    boolExpected : BOOL;
    boolActual : BOOL;
    byteExpected : BYTE;
    byteActual : BYTE;
    dateExpected : DATE;
    dateActual : DATE;
    dateAndTimeExpected : DATE_AND_TIME;
    dateAndTimeActual : DATE_AND_TIME;
    dintExpected : DINT;
    dintActual : DINT;
    dwordExpected : DWORD;
    dwordActual : DWORD;
    intExpected : INT;
    intActual : INT;
    lintExpected : LINT;
    lintActual : LINT;
    lrealExpected : LREAL;
    lrealActual : LREAL;
    ltimeExpected : LTIME;
    ltimeActual : LTIME;
    lwordExpected : LWORD;
    lwordActual : LWORD;
    realExpected : REAL;
    realActual : REAL;
    sintExpected : SINT;
    sintActual : SINT;
    stringExpected : Tc2_System.T_MaxString;
    stringActual : Tc2_System.T_MaxString;
    timeExpected : TIME;
    timeActual : TIME;
    timeOfDayExpected : TIME_OF_DAY;
    timeOfDayActual : TIME_OF_DAY;
    udintExpected : UDINT;
    udintActual : UDINT;
    uintExpected : UINT;
    uintActual : UINT;
    ulintExpected : ULINT;
    ulintActual : ULINT;
    usintExpected : USINT;
    usintActual : USINT;
    wordExpected : WORD;
    wordActual : WORD;
END_VAR
IF GVL_TcUnit.IgnoreCurrentTest OR GVL_TcUnit.CurrentTestIsFinished THEN
    RETURN;
END_IF

AnyComparator(AnyValueOne := Expected,
              AnyValueTwo := Actual);

(* First check whether the input data are any of the standard data types that are supported by TcUnit.
   In this case call the standard Assert-methods for that data. But before doing that we need to make sure
   that both the expected and actual:
   - Have both the same data type
   - Both have the same data size
*)
IF NOT AnyComparator.DataTypesNotEquals AND NOT AnyComparator.DataSizeNotEquals THEN

    (* BOOL *)
    IF UDINT_TO_INT(Expected.TypeClass) = IBaseLibrary.TypeClass.TYPE_BOOL THEN
        Tc2_System.MEMCPY(destAddr := ADR(boolExpected), srcAddr := Expected.pValue, n := SIZEOF(BOOL));
        Tc2_System.MEMCPY(destAddr := ADR(boolActual), srcAddr := Actual.pValue, n := SIZEOF(BOOL));
        AssertEquals_BOOL(Expected := boolExpected, Actual := boolActual, Message := Message);
        RETURN;
    END_IF

    (* BYTE *)
    IF UDINT_TO_INT(Expected.TypeClass) = IBaseLibrary.TypeClass.TYPE_BYTE THEN
        Tc2_System.MEMCPY(destAddr := ADR(byteExpected), srcAddr := Expected.pValue, n := SIZEOF(BYTE));
        Tc2_System.MEMCPY(destAddr := ADR(byteActual), srcAddr := Actual.pValue, n := SIZEOF(BYTE));
        AssertEquals_BYTE(Expected := byteExpected, Actual := byteActual, Message := Message);
        RETURN;
    END_IF

    (* DATE *)
    IF UDINT_TO_INT(Expected.TypeClass) = IBaseLibrary.TypeClass.TYPE_DATE THEN
        Tc2_System.MEMCPY(destAddr := ADR(dateExpected), srcAddr := Expected.pValue, n := SIZEOF(DATE));
        Tc2_System.MEMCPY(destAddr := ADR(dateActual), srcAddr := Actual.pValue, n := SIZEOF(DATE));
        AssertEquals_DATE(Expected := dateExpected, Actual := dateActual, Message := Message);
        RETURN;
    END_IF

    (* DATE_AND_TIME *)
    IF UDINT_TO_INT(Expected.TypeClass) = IBaseLibrary.TypeClass.TYPE_DATEANDTIME THEN
        Tc2_System.MEMCPY(destAddr := ADR(dateAndTimeExpected), srcAddr := Expected.pValue, n := SIZEOF(DATE_AND_TIME));
        Tc2_System.MEMCPY(destAddr := ADR(dateAndTimeActual), srcAddr := Actual.pValue, n := SIZEOF(DATE_AND_TIME));
        AssertEquals_DATE_AND_TIME(Expected := dateAndTimeExpected, Actual := dateAndTimeActual, Message := Message);
        RETURN;
    END_IF

    (* DINT *)
    IF UDINT_TO_INT(Expected.TypeClass) = IBaseLibrary.TypeClass.TYPE_DINT THEN
        Tc2_System.MEMCPY(destAddr := ADR(dintExpected), srcAddr := Expected.pValue, n := SIZEOF(DINT));
        Tc2_System.MEMCPY(destAddr := ADR(dintActual), srcAddr := Actual.pValue, n := SIZEOF(DINT));
        AssertEquals_DINT(Expected := dintExpected, Actual := dintActual, Message := Message);
        RETURN;
    END_IF

    (* DWORD *)
    IF UDINT_TO_INT(Expected.TypeClass) = IBaseLibrary.TypeClass.TYPE_DWORD THEN
        Tc2_System.MEMCPY(destAddr := ADR(dwordExpected), srcAddr := Expected.pValue, n := SIZEOF(DWORD));
        Tc2_System.MEMCPY(destAddr := ADR(dwordActual), srcAddr := Actual.pValue, n := SIZEOF(DWORD));
        AssertEquals_DWORD(Expected := dwordExpected, Actual := dwordActual, Message := Message);
        RETURN;
    END_IF

    (* INT *)
    IF UDINT_TO_INT(Expected.TypeClass) = IBaseLibrary.TypeClass.TYPE_INT THEN
        Tc2_System.MEMCPY(destAddr := ADR(intExpected), srcAddr := Expected.pValue, n := SIZEOF(INT));
        Tc2_System.MEMCPY(destAddr := ADR(intActual), srcAddr := Actual.pValue, n := SIZEOF(INT));
        AssertEquals_INT(Expected := intExpected, Actual := intActual, Message := Message);
        RETURN;
    END_IF

    (* LINT *)
    IF UDINT_TO_INT(Expected.TypeClass) = IBaseLibrary.TypeClass.TYPE_LINT THEN
        Tc2_System.MEMCPY(destAddr := ADR(lintExpected), srcAddr := Expected.pValue, n := SIZEOF(LINT));
        Tc2_System.MEMCPY(destAddr := ADR(lintActual), srcAddr := Actual.pValue, n := SIZEOF(LINT));
        AssertEquals_LINT(Expected := lintExpected, Actual := lintActual, Message := Message);
        RETURN;
    END_IF

    (* LREAL *)
    IF UDINT_TO_INT(Expected.TypeClass) = IBaseLibrary.TypeClass.TYPE_LREAL THEN
        Tc2_System.MEMCPY(destAddr := ADR(lrealExpected), srcAddr := Expected.pValue, n := SIZEOF(LREAL));
        Tc2_System.MEMCPY(destAddr := ADR(lrealActual), srcAddr := Actual.pValue, n := SIZEOF(LREAL));
        AssertEquals_LREAL(Expected := lrealExpected, Actual := lrealActual, Delta := 0.0, Message := Message);
        RETURN;
    END_IF

    (* LTIME *)
    IF UDINT_TO_INT(Expected.TypeClass) = IBaseLibrary.TypeClass.TYPE_LTIME THEN
        Tc2_System.MEMCPY(destAddr := ADR(ltimeExpected), srcAddr := Expected.pValue, n := SIZEOF(LTIME));
        Tc2_System.MEMCPY(destAddr := ADR(ltimeActual), srcAddr := Actual.pValue, n := SIZEOF(LTIME));
        AssertEquals_LTIME(Expected := ltimeExpected, Actual := ltimeActual, Message := Message);
        RETURN;
    END_IF

    (* LWORD *)
    IF UDINT_TO_INT(Expected.TypeClass) = IBaseLibrary.TypeClass.TYPE_LWORD THEN
        Tc2_System.MEMCPY(destAddr := ADR(lwordExpected), srcAddr := Expected.pValue, n := SIZEOF(LWORD));
        Tc2_System.MEMCPY(destAddr := ADR(lwordActual), srcAddr := Actual.pValue, n := SIZEOF(LWORD));
        AssertEquals_LWORD(Expected := lwordExpected, Actual := lwordActual, Message := Message);
        RETURN;
    END_IF

    (* REAL *)
    IF UDINT_TO_INT(Expected.TypeClass) = IBaseLibrary.TypeClass.TYPE_REAL THEN
        Tc2_System.MEMCPY(destAddr := ADR(realExpected), srcAddr := Expected.pValue, n := SIZEOF(REAL));
        Tc2_System.MEMCPY(destAddr := ADR(realActual), srcAddr := Actual.pValue, n := SIZEOF(REAL));
        AssertEquals_REAL(Expected := realExpected, Actual := realActual, Delta := 0.0, Message := Message);
        RETURN;
    END_IF

    (* SINT *)
    IF UDINT_TO_INT(Expected.TypeClass) = IBaseLibrary.TypeClass.TYPE_SINT THEN
        Tc2_System.MEMCPY(destAddr := ADR(sintExpected), srcAddr := Expected.pValue, n := SIZEOF(SINT));
        Tc2_System.MEMCPY(destAddr := ADR(sintActual), srcAddr := Actual.pValue, n := SIZEOF(SINT));
        AssertEquals_SINT(Expected := sintExpected, Actual := sintActual, Message := Message);
        RETURN;
    END_IF

    (* STRING *)
    IF UDINT_TO_INT(Expected.TypeClass) = IBaseLibrary.TypeClass.TYPE_STRING THEN
        Tc2_System.MEMCPY(destAddr := ADR(stringExpected), srcAddr := Expected.pValue, n := DINT_TO_UDINT(Expected.diSize));
        Tc2_System.MEMCPY(destAddr := ADR(stringActual), srcAddr := Actual.pValue, n := DINT_TO_UDINT(Actual.diSize));
        AssertEquals_STRING(Expected := stringExpected, Actual := stringActual, Message := Message);
        RETURN;
    END_IF

    (* TIME *)
    IF UDINT_TO_INT(Expected.TypeClass) = IBaseLibrary.TypeClass.TYPE_TIME THEN
        Tc2_System.MEMCPY(destAddr := ADR(timeExpected), srcAddr := Expected.pValue, n := SIZEOF(TIME));
        Tc2_System.MEMCPY(destAddr := ADR(timeActual), srcAddr := Actual.pValue, n := SIZEOF(TIME));
        AssertEquals_TIME(Expected := timeExpected, Actual := timeActual, Message := Message);
        RETURN;
    END_IF

    (* TIME_OF_DAY *)
    IF UDINT_TO_INT(Expected.TypeClass) = IBaseLibrary.TypeClass.TYPE_TIMEOFDAY THEN
        Tc2_System.MEMCPY(destAddr := ADR(timeOfDayExpected), srcAddr := Expected.pValue, n := SIZEOF(TIME_OF_DAY));
        Tc2_System.MEMCPY(destAddr := ADR(timeOfDayActual), srcAddr := Actual.pValue, n := SIZEOF(TIME_OF_DAY));
        AssertEquals_TIME_OF_DAY(Expected := timeOfDayExpected, Actual := timeOfDayActual, Message := Message);
        RETURN;
    END_IF

    (* UDINT *)
    IF UDINT_TO_INT(Expected.TypeClass) = IBaseLibrary.TypeClass.TYPE_UDINT THEN
        Tc2_System.MEMCPY(destAddr := ADR(udintExpected), srcAddr := Expected.pValue, n := SIZEOF(UDINT));
        Tc2_System.MEMCPY(destAddr := ADR(udintActual), srcAddr := Actual.pValue, n := SIZEOF(UDINT));
        AssertEquals_UDINT(Expected := udintExpected, Actual := udintActual, Message := Message);
        RETURN;
    END_IF

    (* UINT *)
    IF UDINT_TO_INT(Expected.TypeClass) = IBaseLibrary.TypeClass.TYPE_UINT THEN
        Tc2_System.MEMCPY(destAddr := ADR(uintExpected), srcAddr := Expected.pValue, n := SIZEOF(UINT));
        Tc2_System.MEMCPY(destAddr := ADR(uintActual), srcAddr := Actual.pValue, n := SIZEOF(UINT));
        AssertEquals_UINT(Expected := uintExpected, Actual := uintActual, Message := Message);
        RETURN;
    END_IF

    (* ULINT *)
    IF UDINT_TO_INT(Expected.TypeClass) = IBaseLibrary.TypeClass.TYPE_ULINT THEN
        Tc2_System.MEMCPY(destAddr := ADR(ulintExpected), srcAddr := Expected.pValue, n := SIZEOF(ULINT));
        Tc2_System.MEMCPY(destAddr := ADR(ulintActual), srcAddr := Actual.pValue, n := SIZEOF(ULINT));
        AssertEquals_ULINT(Expected := ulintExpected, Actual := ulintActual, Message := Message);
        RETURN;
    END_IF

    (* USINT *)
    IF UDINT_TO_INT(Expected.TypeClass) = IBaseLibrary.TypeClass.TYPE_USINT THEN
        Tc2_System.MEMCPY(destAddr := ADR(usintExpected), srcAddr := Expected.pValue, n := SIZEOF(USINT));
        Tc2_System.MEMCPY(destAddr := ADR(usintActual), srcAddr := Actual.pValue, n := SIZEOF(USINT));
        AssertEquals_USINT(Expected := usintExpected, Actual := usintActual, Message := Message);
        RETURN;
    END_IF

    (* WORD *)
    IF UDINT_TO_INT(Expected.TypeClass) = IBaseLibrary.TypeClass.TYPE_WORD THEN
        Tc2_System.MEMCPY(destAddr := ADR(wordExpected), srcAddr := Expected.pValue, n := SIZEOF(WORD));
        Tc2_System.MEMCPY(destAddr := ADR(wordActual), srcAddr := Actual.pValue, n := SIZEOF(WORD));
        AssertEquals_WORD(Expected := wordExpected, Actual := wordActual, Message := Message);
        RETURN;
    END_IF

END_IF

(* If we've come to this row, it means that the data input is not any of the standard primitive data types, and thus
   we need to do special handling *)
TestInstancePath := AddTestNameToInstancePath(TestInstancePath := FindTestSuiteInstancePath());

IF AnyComparator.DataTypesNotEquals THEN
    ExpectedDataString := Tc2_Standard.CONCAT(STR1 := '(Type class = ', STR2 := F_AnyTypeClassToString((Expected.TypeClass)));
    ExpectedDataString := Tc2_Standard.CONCAT(STR1 := ExpectedDataString, STR2 := ')');
    ActualDataString := Tc2_Standard.CONCAT(STR1 := '(Type class = ', STR2 := F_AnyTypeClassToString(Actual.TypeClass));
    ActualDataString := Tc2_Standard.CONCAT(STR1 := ActualDataString, STR2 := ')');
ELSIF AnyComparator.DataSizeNotEquals THEN
    ExpectedDataString := Tc2_Standard.CONCAT(STR1 := '(Data size = ', STR2 := DINT_TO_STRING(Expected.diSize));
    ExpectedDataString := Tc2_Standard.CONCAT(STR1 := ExpectedDataString, STR2 := ')');
    ActualDataString := Tc2_Standard.CONCAT(STR1 := '(Data size = ', STR2 := DINT_TO_STRING(Actual.diSize));
    ActualDataString := Tc2_Standard.CONCAT(STR1 := ActualDataString, STR2 := ')');
ELSIF AnyComparator.DataContentNotEquals THEN
    FOR Count := 0 TO MIN(Expected.diSize-1, 38) BY 1 DO // One byte will equal two characters (example: 255 = 0xff, 1 = 0x01)
        ExpectedDataString := Tc2_Standard.CONCAT(STR1 := ExpectedDataString,
                                                  STR2 := Tc2_Utilities.BYTE_TO_HEXSTR(in := Expected.pValue[Count],
                                                                                       iPrecision := 2,
                                                                                       bLoCase := FALSE));
    END_FOR
    ExpectedDataString := Tc2_Standard.CONCAT(STR1 := '0x', STR2 := ExpectedDataString);

    FOR Count := 0 TO MIN(Actual.diSize-1, 38) BY 1 DO // One byte will equal two characters (example: 255 = 0xff, 1 = 0x01)
        ActualDataString := Tc2_Standard.CONCAT(STR1 := ActualDataString,
                                                STR2 := Tc2_Utilities.BYTE_TO_HEXSTR(in := Actual.pValue[Count],
                                                                                     iPrecision := 2,
                                                                                     bLoCase := FALSE));
    END_FOR
    ActualDataString := Tc2_Standard.CONCAT(STR1 := '0x', STR2 := ActualDataString);
END_IF

IF (AnyComparator.DataTypesNotEquals OR AnyComparator.DataSizeNotEquals OR AnyComparator.DataContentNotEquals) THEN
    AssertResults.ReportResult(Expected := Expected,
                               Actual := Actual,
                               Message := Message,
                               TestInstancePath := TestInstancePath,
                               AlreadyReported => AlreadyReported);
END_IF

IF NOT AlreadyReported AND (AnyComparator.DataTypesNotEquals OR AnyComparator.DataSizeNotEquals OR AnyComparator.DataContentNotEquals) THEN
    SetTestFailed();

    AssertMessageFormatter.LogAssertFailure(Expected := ExpectedDataString,
                                            Actual := ActualDataString,
                                            Message := Message,
                                            TestInstancePath := TestInstancePath);
END_IF
END_METHOD

(*
    Asserts that two BOOLs are equal. If they are not, an assertion error is created.
*)
METHOD PUBLIC AssertEquals_BOOL
VAR_INPUT
    Expected : BOOL; // BOOL expected value
    Actual : BOOL; // BOOL actual value
    Message : Tc2_System.T_MaxString; // The identifying message for the assertion error
END_VAR
VAR
    AlreadyReported : BOOL;
    TestInstancePath : Tc2_System.T_MaxString;
END_VAR
IF GVL_TcUnit.IgnoreCurrentTest OR GVL_TcUnit.CurrentTestIsFinished THEN
    RETURN;
END_IF

TestInstancePath := AddTestNameToInstancePath(TestInstancePath := FindTestSuiteInstancePath());

IF Expected <> Actual THEN
    AssertResults.ReportResult(Expected := Expected,
                               Actual := Actual,
                               Message := Message,
                               TestInstancePath := TestInstancePath,
                               AlreadyReported => AlreadyReported);
END_IF                               

IF NOT AlreadyReported AND Expected <> Actual THEN
    SetTestFailed();

    AssertMessageFormatter.LogAssertFailure(Expected := BOOL_TO_STRING(Expected),
                                            Actual := BOOL_TO_STRING(Actual),
                                            Message := Message,
                                            TestInstancePath := TestInstancePath);
END_IF
END_METHOD

(*
    Asserts that two BYTEs are equal. If they are not, an assertion error is created.
*)
METHOD PUBLIC AssertEquals_BYTE
VAR_INPUT
    Expected : BYTE; // BYTE expected value
    Actual : BYTE; // BYTE actual value
    Message : Tc2_System.T_MaxString; // The identifying message for the assertion error
END_VAR
VAR
    TestInstancePath : Tc2_System.T_MaxString;
    AlreadyReported : BOOL;
END_VAR
IF GVL_TcUnit.IgnoreCurrentTest OR GVL_TcUnit.CurrentTestIsFinished THEN
    RETURN;
END_IF

TestInstancePath := AddTestNameToInstancePath(TestInstancePath := FindTestSuiteInstancePath());

IF Expected <> Actual THEN
    AssertResults.ReportResult(Expected := Expected,
                               Actual := Actual,
                               Message := Message,
                               TestInstancePath := TestInstancePath,
                               AlreadyReported => AlreadyReported);
END_IF

IF NOT AlreadyReported AND Expected <> Actual THEN
    SetTestFailed();

    AssertMessageFormatter.LogAssertFailure(Expected := Tc2_Standard.CONCAT(
                                                       STR1 := '0x',
                                                       STR2 := Tc2_Utilities.BYTE_TO_HEXSTR(in := Expected,
                                                                                            iPrecision := 2,
                                                                                            bLoCase := FALSE)),
                                            Actual := Tc2_Standard.CONCAT(
                                                       STR1 := '0x',
                                                       STR2 := Tc2_Utilities.BYTE_TO_HEXSTR(in := Actual,
                                                                                            iPrecision := 2,
                                                                                            bLoCase := FALSE)),
                                            Message := Message,
                                            TestInstancePath := TestInstancePath);
END_IF
END_METHOD

(*
    Asserts that two DATEs are equal. If they are not, an assertion error is created.
*)
METHOD PUBLIC AssertEquals_DATE
VAR_INPUT
    Expected : DATE; // DATE expected value
    Actual : DATE; // DATE actual value
    Message : Tc2_System.T_MaxString; // The identifying message for the assertion error
END_VAR
VAR
    TestInstancePath : Tc2_System.T_MaxString;
    AlreadyReported : BOOL;
END_VAR
IF GVL_TcUnit.IgnoreCurrentTest OR GVL_TcUnit.CurrentTestIsFinished THEN
    RETURN;
END_IF

TestInstancePath := AddTestNameToInstancePath(TestInstancePath := FindTestSuiteInstancePath());

IF Expected <> Actual THEN
    AssertResults.ReportResult(Expected := Expected,
                               Actual := Actual,
                               Message := Message,
                               TestInstancePath := TestInstancePath,
                               AlreadyReported => AlreadyReported);
END_IF

IF NOT AlreadyReported AND Expected <> Actual THEN
    SetTestFailed();

    AssertMessageFormatter.LogAssertFailure(Expected := DATE_TO_STRING(Expected),
                                            Actual := DATE_TO_STRING(Actual),
                                            Message := Message,
                                            TestInstancePath := TestInstancePath);
END_IF
END_METHOD

(*
    Asserts that two DATE_AND_TIMEs are equal. If they are not, an assertion error is created.
*)
METHOD PUBLIC AssertEquals_DATE_AND_TIME
VAR_INPUT
    Expected : DATE_AND_TIME; // DATE_AND_TIME expected value
    Actual : DATE_AND_TIME; // DATE_AND_TIME actual value
    Message : Tc2_System.T_MaxString; // The identifying message for the assertion error
END_VAR
VAR
    TestInstancePath : Tc2_System.T_MaxString;
    AlreadyReported : BOOL;
END_VAR
IF GVL_TcUnit.IgnoreCurrentTest OR GVL_TcUnit.CurrentTestIsFinished THEN
    RETURN;
END_IF

TestInstancePath := AddTestNameToInstancePath(TestInstancePath := FindTestSuiteInstancePath());

IF Expected <> Actual THEN
    AssertResults.ReportResult(Expected := Expected,
                               Actual := Actual,
                               Message := Message,
                               TestInstancePath := TestInstancePath,
                               AlreadyReported => AlreadyReported);
END_IF

IF NOT AlreadyReported AND Expected <> Actual THEN
    SetTestFailed();

    AssertMessageFormatter.LogAssertFailure(Expected := DT_TO_STRING(Expected),
                                            Actual := DT_TO_STRING(Actual),
                                            Message := Message,
                                            TestInstancePath := TestInstancePath);
END_IF
END_METHOD

(*
    Asserts that two DINTs are equal. If they are not, an assertion error is created.
*)
METHOD PUBLIC AssertEquals_DINT
VAR_INPUT
    Expected : DINT; // DINT expected value
    Actual : DINT; // DINT actual value
    Message : Tc2_System.T_MaxString; // The identifying message for the assertion error
END_VAR
VAR
    TestInstancePath : Tc2_System.T_MaxString;
    AlreadyReported : BOOL;
END_VAR
IF GVL_TcUnit.IgnoreCurrentTest OR GVL_TcUnit.CurrentTestIsFinished THEN
    RETURN;
END_IF

TestInstancePath := AddTestNameToInstancePath(TestInstancePath := FindTestSuiteInstancePath());

IF Expected <> Actual THEN
    AssertResults.ReportResult(Expected := Expected,
                               Actual := Actual,
                               Message := Message,
                               TestInstancePath := TestInstancePath,
                               AlreadyReported => AlreadyReported);
END_IF

IF NOT AlreadyReported AND Expected <> Actual THEN
    SetTestFailed();

    AssertMessageFormatter.LogAssertFailure(Expected := DINT_TO_STRING(Expected),
                                            Actual := DINT_TO_STRING(Actual),
                                            Message := Message,
                                            TestInstancePath := TestInstancePath);
END_IF
END_METHOD

(*
    Asserts that two DWORDs are equal. If they are not, an assertion error is created.
*)
METHOD PUBLIC AssertEquals_DWORD
VAR_INPUT
    Expected : DWORD; // DWORD expected value
    Actual : DWORD; // DWORD actual value
    Message : Tc2_System.T_MaxString; // The identifying message for the assertion error
END_VAR
VAR
    TestInstancePath : Tc2_System.T_MaxString;
    AlreadyReported : BOOL;
END_VAR
IF GVL_TcUnit.IgnoreCurrentTest OR GVL_TcUnit.CurrentTestIsFinished THEN
    RETURN;
END_IF

TestInstancePath := AddTestNameToInstancePath(TestInstancePath := FindTestSuiteInstancePath());

IF Expected <> Actual THEN
    AssertResults.ReportResult(Expected := Expected,
                               Actual := Actual,
                               Message := Message,
                               TestInstancePath := TestInstancePath,
                               AlreadyReported => AlreadyReported);
END_IF

IF NOT AlreadyReported AND Expected <> Actual THEN
    SetTestFailed();

    AssertMessageFormatter.LogAssertFailure(Expected := Tc2_Standard.CONCAT(
                                                            STR1 := '0x',
                                                            STR2 := Tc2_Utilities.DWORD_TO_HEXSTR(in := Expected,
                                                                                                  iPrecision := 8,
                                                                                                  bLoCase := FALSE)),
                                            Actual := Tc2_Standard.CONCAT(
                                                           STR1 := '0x',
                                                           STR2 := Tc2_Utilities.DWORD_TO_HEXSTR(in := Actual,
                                                                                                 iPrecision := 8,
                                                                                                 bLoCase := FALSE)),
                                            Message := Message,
                                            TestInstancePath := TestInstancePath);
END_IF
END_METHOD

(*
    Asserts that two INTs are equal. If they are not, an assertion error is created.
*)
METHOD PUBLIC AssertEquals_INT
VAR_INPUT
    Expected : INT; // INT expected value
    Actual : INT; // INT actual value
    Message : Tc2_System.T_MaxString; // The identifying message for the assertion error
END_VAR
VAR
    TestInstancePath : Tc2_System.T_MaxString;
    AlreadyReported : BOOL;
END_VAR
IF GVL_TcUnit.IgnoreCurrentTest OR GVL_TcUnit.CurrentTestIsFinished THEN
    RETURN;
END_IF

TestInstancePath := AddTestNameToInstancePath(TestInstancePath := FindTestSuiteInstancePath());

IF Expected <> Actual THEN
    AssertResults.ReportResult(Expected := Expected,
                               Actual := Actual,
                               Message := Message,
                               TestInstancePath := TestInstancePath,
                               AlreadyReported => AlreadyReported);
END_IF

IF NOT AlreadyReported AND Expected <> Actual THEN
    SetTestFailed();

    AssertMessageFormatter.LogAssertFailure(Expected := INT_TO_STRING(Expected),
                                            Actual := INT_TO_STRING(Actual),
                                            Message := Message,
                                            TestInstancePath := TestInstancePath);
END_IF
END_METHOD

(*
    Asserts that two LINTs are equal. If they are not, an assertion error is created.
*)
METHOD PUBLIC AssertEquals_LINT
VAR_INPUT
    Expected : LINT; // LINT expected value
    Actual : LINT; // LINT actual value
    Message : Tc2_System.T_MaxString; // The identifying message for the assertion error
END_VAR
VAR
    TestInstancePath : Tc2_System.T_MaxString;
    AlreadyReported : BOOL;
END_VAR
IF GVL_TcUnit.IgnoreCurrentTest OR GVL_TcUnit.CurrentTestIsFinished THEN
    RETURN;
END_IF

TestInstancePath := AddTestNameToInstancePath(TestInstancePath := FindTestSuiteInstancePath());

IF Expected <> Actual THEN
    AssertResults.ReportResult(Expected := Expected,
                               Actual := Actual,
                               Message := Message,
                               TestInstancePath := TestInstancePath,
                               AlreadyReported => AlreadyReported);
END_IF

IF NOT AlreadyReported AND Expected <> Actual THEN
    SetTestFailed();

    AssertMessageFormatter.LogAssertFailure(Expected := LINT_TO_STRING(Expected),
                                            Actual := LINT_TO_STRING(Actual),
                                            Message := Message,
                                            TestInstancePath := TestInstancePath);
END_IF
END_METHOD

(*
    Asserts that two LREALs are equal to within a positive delta. If they are not, an assertion error is created.
*)
METHOD PUBLIC AssertEquals_LREAL
VAR_INPUT
    Expected : LREAL; // LREAL expected value
    Actual : LREAL; // LREAL actual value
    Delta : LREAL; // The maximum delta between the absolute value of expected and actual for which both numbers are still considered equal
    Message : Tc2_System.T_MaxString; // The identifying message for the assertion error
END_VAR
VAR
    TestInstancePath : Tc2_System.T_MaxString;
    AlreadyReported : BOOL;
END_VAR
IF GVL_TcUnit.IgnoreCurrentTest OR GVL_TcUnit.CurrentTestIsFinished THEN
    RETURN;
END_IF

TestInstancePath := AddTestNameToInstancePath(TestInstancePath := FindTestSuiteInstancePath());

IF ABS(Expected - Actual) > Delta THEN
    AssertResults.ReportResult(Expected := Expected,
                               Actual := Actual,
                               Message := Message,
                               TestInstancePath := TestInstancePath,
                               AlreadyReported => AlreadyReported);
END_IF

IF NOT AlreadyReported AND ABS(Expected - Actual) > Delta THEN
    SetTestFailed();

    AssertMessageFormatter.LogAssertFailure(Expected := LREAL_TO_STRING(Expected),
                                            Actual := LREAL_TO_STRING(Actual),
                                            Message := Message,
                                            TestInstancePath := TestInstancePath);
END_IF
END_METHOD

(*
    Asserts that two LTIMEs are equal. If they are not, an assertion error is created.
*)
METHOD PUBLIC AssertEquals_LTIME
VAR_INPUT
    Expected : LTIME; // LTIME expected value
    Actual : LTIME; // LTIME actual value
    Message : Tc2_System.T_MaxString; // The identifying message for the assertion error
END_VAR
VAR
    TestInstancePath : Tc2_System.T_MaxString;
    AlreadyReported : BOOL;
END_VAR
IF GVL_TcUnit.IgnoreCurrentTest OR GVL_TcUnit.CurrentTestIsFinished THEN
    RETURN;
END_IF

TestInstancePath := AddTestNameToInstancePath(TestInstancePath := FindTestSuiteInstancePath());

IF Expected <> Actual THEN
    AssertResults.ReportResult(Expected := Expected,
                               Actual := Actual,
                               Message := Message,
                               TestInstancePath := TestInstancePath,
                               AlreadyReported => AlreadyReported);
END_IF

IF NOT AlreadyReported AND Expected <> Actual THEN
    SetTestFailed();

    AssertMessageFormatter.LogAssertFailure(Expected := LTIME_TO_STRING(Expected),
                                            Actual := LTIME_TO_STRING(Actual),
                                            Message := Message,
                                            TestInstancePath := TestInstancePath);
END_IF
END_METHOD

(*
    Asserts that two LWORDs are equal. If they are not, an assertion error is created.
*)
METHOD PUBLIC AssertEquals_LWORD
VAR_INPUT
    Expected : LWORD; // LWORD expected value
    Actual : LWORD; // LWORD actual value
    Message : Tc2_System.T_MaxString; // The identifying message for the assertion error
END_VAR
VAR
    TestInstancePath : Tc2_System.T_MaxString;
    AlreadyReported : BOOL;
END_VAR
IF GVL_TcUnit.IgnoreCurrentTest OR GVL_TcUnit.CurrentTestIsFinished THEN
    RETURN;
END_IF

TestInstancePath := AddTestNameToInstancePath(TestInstancePath := FindTestSuiteInstancePath());

IF Expected <> Actual THEN
    AssertResults.ReportResult(Expected := Expected,
                               Actual := Actual,
                               Message := Message,
                               TestInstancePath := TestInstancePath,
                               AlreadyReported => AlreadyReported);
END_IF

IF NOT AlreadyReported AND Expected <> Actual THEN
    SetTestFailed();

    AssertMessageFormatter.LogAssertFailure(Expected := Tc2_Standard.CONCAT(
                                                            STR1 := '0x',
                                                            STR2 := Tc2_Utilities.LWORD_TO_HEXSTR(in := Expected,
                                                                                                  iPrecision := 16,
                                                                                                  bLoCase := FALSE)),
                                            Actual := Tc2_Standard.CONCAT(
                                                            STR1 := '0x',
                                                            STR2 := Tc2_Utilities.LWORD_TO_HEXSTR(in := Actual,
                                                                                                  iPrecision := 16,
                                                                                                  bLoCase := FALSE)),
                                            Message := Message,
                                            TestInstancePath := TestInstancePath);
END_IF
END_METHOD

(*
    Asserts that two REALs are equal to within a positive delta. If they are not, an assertion error is created.
*)
METHOD PUBLIC AssertEquals_REAL
VAR_INPUT
    Expected : REAL; // REAL expected value
    Actual : REAL; // REAL actual value
    Delta : REAL;  // The maximum delta between the absolute value of expected and actual for which both numbers are still considered equal
    Message : Tc2_System.T_MaxString; // The identifying message for the assertion error
END_VAR
VAR
    TestInstancePath : Tc2_System.T_MaxString;
    AlreadyReported : BOOL;
END_VAR
IF GVL_TcUnit.IgnoreCurrentTest OR GVL_TcUnit.CurrentTestIsFinished THEN
    RETURN;
END_IF

TestInstancePath := AddTestNameToInstancePath(TestInstancePath := FindTestSuiteInstancePath());

IF ABS(Expected - Actual) > Delta THEN
    AssertResults.ReportResult(Expected := Expected,
                               Actual := Actual,
                               Message := Message,
                               TestInstancePath := TestInstancePath,
                               AlreadyReported => AlreadyReported);
END_IF

IF NOT AlreadyReported AND ABS(Expected - Actual) > Delta THEN
    SetTestFailed();

    AssertMessageFormatter.LogAssertFailure(Expected := REAL_TO_STRING(Expected),
                                            Actual := REAL_TO_STRING(Actual),
                                            Message := Message,
                                            TestInstancePath := TestInstancePath);
END_IF
END_METHOD

(*
    Asserts that two SINTs are equal. If they are not, an assertion error is created.
*)
METHOD PUBLIC AssertEquals_SINT
VAR_INPUT
    Expected : SINT; // SINT expected value
    Actual : SINT; // SINT actual value
    Message : Tc2_System.T_MaxString; // The identifying message for the assertion error
END_VAR
VAR
    TestInstancePath : Tc2_System.T_MaxString;
    AlreadyReported : BOOL;
END_VAR
IF GVL_TcUnit.IgnoreCurrentTest OR GVL_TcUnit.CurrentTestIsFinished THEN
    RETURN;
END_IF

TestInstancePath := AddTestNameToInstancePath(TestInstancePath := FindTestSuiteInstancePath());

IF Expected <> Actual THEN
    AssertResults.ReportResult(Expected := Expected,
                               Actual := Actual,
                               Message := Message,
                               TestInstancePath := TestInstancePath,
                               AlreadyReported => AlreadyReported);
END_IF

IF NOT AlreadyReported AND Expected <> Actual THEN
    SetTestFailed();

    AssertMessageFormatter.LogAssertFailure(Expected := SINT_TO_STRING(Expected),
                                            Actual := SINT_TO_STRING(Actual),
                                            Message := Message,
                                            TestInstancePath := TestInstancePath);
END_IF
END_METHOD

(*
    Asserts that two STRINGs are equal. If they are not, an assertion error is created.
*)
METHOD PUBLIC AssertEquals_STRING
VAR_INPUT
    Expected : Tc2_System.T_MaxString; // STRING expected value
    Actual : Tc2_System.T_MaxString; // STRING actual value
    Message : Tc2_System.T_MaxString; // The identifying message for the assertion error
END_VAR
VAR
    TestInstancePath : Tc2_System.T_MaxString;
    AlreadyReported : BOOL;
END_VAR
IF GVL_TcUnit.IgnoreCurrentTest OR GVL_TcUnit.CurrentTestIsFinished THEN
    RETURN;
END_IF

TestInstancePath := AddTestNameToInstancePath(TestInstancePath := FindTestSuiteInstancePath());

IF (Tc2_Standard.LEN(STR := Expected) <> Tc2_Standard.LEN(STR := Actual) OR (Expected <> Actual)) THEN
    AssertResults.ReportResult(Expected := Expected,
                               Actual := Actual,
                               Message := Message,
                               TestInstancePath := TestInstancePath,
                               AlreadyReported => AlreadyReported);
END_IF

IF NOT AlreadyReported AND (Tc2_Standard.LEN(STR := Expected) <> Tc2_Standard.LEN(STR := Actual) OR (Expected <> Actual)) THEN
    SetTestFailed();

    AssertMessageFormatter.LogAssertFailure(Expected := Expected,
                                            Actual := Actual,
                                            Message := Message,
                                            TestInstancePath := TestInstancePath);
END_IF
END_METHOD

(*
    Asserts that two TIMEs are equal. If they are not, an assertion error is created.
*)
METHOD PUBLIC AssertEquals_TIME
VAR_INPUT
    Expected : TIME; // TIME expected value
    Actual : TIME; // TIME actual value
    Message : Tc2_System.T_MaxString; // The identifying message for the assertion error
END_VAR
VAR
    TestInstancePath : Tc2_System.T_MaxString;
    AlreadyReported : BOOL;
END_VAR
IF GVL_TcUnit.IgnoreCurrentTest OR GVL_TcUnit.CurrentTestIsFinished THEN
    RETURN;
END_IF

TestInstancePath := AddTestNameToInstancePath(TestInstancePath := FindTestSuiteInstancePath());

IF Expected <> Actual THEN
    AssertResults.ReportResult(Expected := Expected,
                               Actual := Actual,
                               Message := Message,
                               TestInstancePath := TestInstancePath,
                               AlreadyReported => AlreadyReported);
END_IF

IF NOT AlreadyReported AND Expected <> Actual THEN
    SetTestFailed();

    AssertMessageFormatter.LogAssertFailure(Expected := TIME_TO_STRING(Expected),
                                            Actual := TIME_TO_STRING(Actual),
                                            Message := Message,
                                            TestInstancePath := TestInstancePath);
END_IF
END_METHOD

(*
    Asserts that two TIME_OF_DAYs are equal. If they are not, an assertion error is created.
*)
METHOD PUBLIC AssertEquals_TIME_OF_DAY
VAR_INPUT
    Expected : TIME_OF_DAY; // TIME_OF_DAY expected value
    Actual : TIME_OF_DAY; // TIME_OF_DAY actual value
    Message : Tc2_System.T_MaxString; // The identifying message for the assertion error
END_VAR
VAR
    TestInstancePath : Tc2_System.T_MaxString;
    AlreadyReported : BOOL;
END_VAR
IF GVL_TcUnit.IgnoreCurrentTest OR GVL_TcUnit.CurrentTestIsFinished THEN
    RETURN;
END_IF

TestInstancePath := AddTestNameToInstancePath(TestInstancePath := FindTestSuiteInstancePath());

IF Expected <> Actual THEN
    AssertResults.ReportResult(Expected := Expected,
                               Actual := Actual,
                               Message := Message,
                               TestInstancePath := TestInstancePath,
                               AlreadyReported => AlreadyReported);
END_IF

IF NOT AlreadyReported AND Expected <> Actual THEN
    SetTestFailed();

    AssertMessageFormatter.LogAssertFailure(Expected := TOD_TO_STRING(Expected),
                                            Actual := TOD_TO_STRING(Actual),
                                            Message := Message,
                                            TestInstancePath := TestInstancePath);
END_IF
END_METHOD

(*
    Asserts that two UDINTs are equal. If they are not, an assertion error is created.
*)
METHOD PUBLIC AssertEquals_UDINT
VAR_INPUT
    Expected : UDINT; // UDINT expected value
    Actual : UDINT; // UDINT actual value
    Message : Tc2_System.T_MaxString; // The identifying message for the assertion error
END_VAR
VAR
    TestInstancePath : Tc2_System.T_MaxString;
    AlreadyReported : BOOL;
END_VAR
IF GVL_TcUnit.IgnoreCurrentTest OR GVL_TcUnit.CurrentTestIsFinished THEN
    RETURN;
END_IF

TestInstancePath := AddTestNameToInstancePath(TestInstancePath := FindTestSuiteInstancePath());

IF Expected <> Actual THEN
    AssertResults.ReportResult(Expected := Expected,
                               Actual := Actual,
                               Message := Message,
                               TestInstancePath := TestInstancePath,
                               AlreadyReported => AlreadyReported);
END_IF

IF NOT AlreadyReported AND Expected <> Actual THEN
    SetTestFailed();

    AssertMessageFormatter.LogAssertFailure(Expected := UDINT_TO_STRING(Expected),
                                            Actual := UDINT_TO_STRING(Actual),
                                            Message := Message,
                                            TestInstancePath := TestInstancePath);
END_IF
END_METHOD

(*
    Asserts that two UINTs are equal. If they are not, an assertion error is created.
*)
METHOD PUBLIC AssertEquals_UINT
VAR_INPUT
    Expected : UINT; // UINT expected value
    Actual : UINT; // UINT actual value
    Message : Tc2_System.T_MaxString; // The identifying message for the assertion error
END_VAR
VAR
    TestInstancePath : Tc2_System.T_MaxString;
    AlreadyReported : BOOL;
END_VAR
IF GVL_TcUnit.IgnoreCurrentTest OR GVL_TcUnit.CurrentTestIsFinished THEN
    RETURN;
END_IF

TestInstancePath := AddTestNameToInstancePath(TestInstancePath := FindTestSuiteInstancePath());

IF Expected <> Actual THEN
    AssertResults.ReportResult(Expected := Expected,
                               Actual := Actual,
                               Message := Message,
                               TestInstancePath := TestInstancePath,
                               AlreadyReported => AlreadyReported);
END_IF

IF NOT AlreadyReported AND Expected <> Actual THEN
    SetTestFailed();

    AssertMessageFormatter.LogAssertFailure(Expected := UINT_TO_STRING(Expected),
                                            Actual := UINT_TO_STRING(Actual),
                                            Message := Message,
                                            TestInstancePath := TestInstancePath);
END_IF
END_METHOD

(*
    Asserts that two ULINTs are equal. If they are not, an assertion error is created.
*)
METHOD PUBLIC AssertEquals_ULINT
VAR_INPUT
    Expected : ULINT; // ULINT expected value
    Actual : ULINT; // ULINT actual value
    Message : Tc2_System.T_MaxString; // The identifying message for the assertion error
END_VAR
VAR
    TestInstancePath : Tc2_System.T_MaxString;
    AlreadyReported : BOOL;
END_VAR
IF GVL_TcUnit.IgnoreCurrentTest OR GVL_TcUnit.CurrentTestIsFinished THEN
    RETURN;
END_IF

TestInstancePath := AddTestNameToInstancePath(TestInstancePath := FindTestSuiteInstancePath());

IF Expected <> Actual THEN
    AssertResults.ReportResult(Expected := Expected,
                               Actual := Actual,
                               Message := Message,
                               TestInstancePath := TestInstancePath,
                               AlreadyReported => AlreadyReported);
END_IF

IF NOT AlreadyReported AND Expected <> Actual THEN
    SetTestFailed();

    AssertMessageFormatter.LogAssertFailure(Expected := ULINT_TO_STRING(Expected),
                                            Actual := ULINT_TO_STRING(Actual),
                                            Message := Message,
                                            TestInstancePath := TestInstancePath);
END_IF
END_METHOD

(*
    Asserts that two USINTs are equal. If they are not, an assertion error is created.
*)
METHOD PUBLIC AssertEquals_USINT
VAR_INPUT
    Expected : USINT; // USINT expected value
    Actual : USINT; // USINT actual value
    Message : Tc2_System.T_MaxString; // The identifying message for the assertion error
END_VAR
VAR
    AlreadyReported : BOOL;
    TestInstancePath : Tc2_System.T_MaxString;
END_VAR
IF GVL_TcUnit.IgnoreCurrentTest OR GVL_TcUnit.CurrentTestIsFinished THEN
    RETURN;
END_IF

TestInstancePath := AddTestNameToInstancePath(TestInstancePath := FindTestSuiteInstancePath());

IF Expected <> Actual THEN
    AssertResults.ReportResult(Expected := Expected,
                               Actual := Actual,
                               Message := Message,
                               TestInstancePath := TestInstancePath,
                               AlreadyReported => AlreadyReported);
END_IF

IF NOT AlreadyReported AND Expected <> Actual THEN
    SetTestFailed();

    AssertMessageFormatter.LogAssertFailure(Expected := USINT_TO_STRING(Expected),
                                            Actual := USINT_TO_STRING(Actual),
                                            Message := Message,
                                            TestInstancePath := TestInstancePath);
END_IF
END_METHOD

(*
    Asserts that two WORDs are equal. If they are not, an assertion error is created.
*)
METHOD PUBLIC AssertEquals_WORD
VAR_INPUT
    Expected : WORD; // WORD expected value
    Actual : WORD; // WORD actual value
    Message : Tc2_System.T_MaxString; // The identifying message for the assertion error
END_VAR
VAR
    TestInstancePath : Tc2_System.T_MaxString;
    AlreadyReported : BOOL;
END_VAR
IF GVL_TcUnit.IgnoreCurrentTest OR GVL_TcUnit.CurrentTestIsFinished THEN
    RETURN;
END_IF

TestInstancePath := AddTestNameToInstancePath(TestInstancePath := FindTestSuiteInstancePath());

IF Expected <> Actual THEN
    AssertResults.ReportResult(Expected := Expected,
                               Actual := Actual,
                               Message := Message,
                               TestInstancePath := TestInstancePath,
                               AlreadyReported => AlreadyReported);
END_IF

IF NOT AlreadyReported AND Expected <> Actual THEN
    SetTestFailed();

    AssertMessageFormatter.LogAssertFailure(Expected := Tc2_Standard.CONCAT(
                                                            STR1 := '0x',
                                                            STR2 := Tc2_Utilities.WORD_TO_HEXSTR(in := Expected,
                                                                                                 iPrecision := 4,
                                                                                                 bLoCase := FALSE)),
                                            Actual := Tc2_Standard.CONCAT(
                                                            STR1 := '0x',
                                                            STR2 := Tc2_Utilities.WORD_TO_HEXSTR(in := Actual,
                                                                                                 iPrecision := 4,
                                                                                                 bLoCase := FALSE)),
                                            Message := Message,
                                            TestInstancePath := TestInstancePath);
END_IF
END_METHOD

(*
    Asserts that a condition is false. If it is not, an assertion error is created.
*)
METHOD PUBLIC AssertFalse
VAR_INPUT
    Condition : BOOL; // Condition to be checked
    Message : Tc2_System.T_MaxString; // The identifying message for the assertion error
END_VAR
AssertEquals_BOOL(Expected := FALSE, Actual := Condition, Message := Message);
END_METHOD

(*
    Asserts that a condition is true. If it is not, an assertion error is created.
*)
METHOD PUBLIC AssertTrue
VAR_INPUT
    Condition : BOOL; // Condition to be checked
    Message : Tc2_System.T_MaxString; // The identifying message for the assertion error
END_VAR
AssertEquals_BOOL(Expected := TRUE, Actual := Condition, Message := Message);
END_METHOD

METHOD FB_init : BOOL
VAR_INPUT
    bInitRetains : BOOL; // if TRUE, the retain variables are initialized (warm start / cold start)
    bInCopyCode : BOOL;  // if TRUE, the instance afterwards gets moved into the copy code (online change)
END_VAR
GVL_TcUnit.NumberOfInitializedTestSuites := GVL_TcUnit.NumberOfInitializedTestSuites + 1;    
GVL_TcUnit.TestSuiteAddresses[GVL_TcUnit.NumberOfInitializedTestSuites] := THIS;
END_METHOD

(* Searches for the instance path of the calling function block *)
METHOD PRIVATE FindTestSuiteInstancePath : Tc2_System.T_MaxString
FindTestSuiteInstancePath := GetInstancePath();
END_METHOD

METHOD PUBLIC GetInstancePath : Tc2_System.T_MaxString
GetInstancePath := InstancePath;
END_METHOD

METHOD PUBLIC GetNumberOfFailedTests : UINT
VAR
    Counter : UINT;
    FailedTestsCount : UINT;
END_VAR
IF NumberOfTests > 0 THEN
    FOR Counter := 1 TO GetNumberOfTests() BY 1 DO
        IF Tests[Counter].IsFailed() THEN
            FailedTestsCount := FailedTestsCount + 1;
        END_IF
    END_FOR
END_IF

GetNumberOfFailedTests := FailedTestsCount;
END_METHOD

METHOD PUBLIC GetNumberOfSuccessfulTests : UINT
GetNumberOfSuccessfulTests := GetNumberOfTests() - GetNumberOfFailedTests();
END_METHOD

METHOD PUBLIC GetNumberOfTests : UINT
GetNumberOfTests := NumberOfTests;
END_METHOD

METHOD PUBLIC IsTestFinished : BOOL
VAR_INPUT
    TestName : Tc2_System.T_MaxString;
END_VAR
VAR
    IteratorCounter : UINT;
END_VAR
IsTestFinished := FALSE;
IF NumberOfTests > 0 THEN
    FOR IteratorCounter := 1 TO NumberOfTests BY 1 DO
        IF Tests[IteratorCounter].GetName() = TestName THEN
            IsTestFinished := Tests[IteratorCounter].IsFinished();
            RETURN;
        END_IF
    END_FOR
END_IF
END_METHOD

METHOD PUBLIC SetTestFailed
VAR
    IteratorCounter : UINT;
END_VAR
IF NumberOfTests > 0 THEN
    FOR IteratorCounter := 1 TO NumberOfTests BY 1 DO
        IF Tests[IteratorCounter].GetName() = GVL_TcUnit.CurrentTestNameBeingCalled THEN
            Tests[IteratorCounter].SetFailed();
        END_IF
    END_FOR
END_IF
END_METHOD

(* Marks the test as finished in this testsuite.
   Returns TRUE if test was found, and FALSE if a test with this name was not found in this testsuite
*)
METHOD PUBLIC SetTestFinished : BOOL;
VAR_INPUT
    TestName : Tc2_System.T_MaxString;
END_VAR
VAR
    IteratorCounter : UINT;
END_VAR
IF NumberOfTests > 0 THEN
    FOR IteratorCounter := 1 TO NumberOfTests BY 1 DO
        IF Tests[IteratorCounter].GetName() = TestName THEN
            Tests[IteratorCounter].SetFinished();
            SetTestFinished := TRUE;
            RETURN;
        END_IF
    SetTestFinished := FALSE;
    END_FOR
END_IF
END_METHOD

END_FUNCTION_BLOCK
